PROGRAM MAIN
VAR
	a:BOOL;
	b:INT;
END_VAR

a:=TRUE;

END_PROGRAM

(* stored: Version 1.1.0.1, ProductVersion 3.1.4024.6
   POU MAIN: Id {4b4f205d-eb1e-4370-985b-8b97e2c05bd2}, SpecialFunc None *)
